TYPE U_Union :
UNION
	INT_	: INT;
	BOOL_	: BOOL;
	UDINT_	: UDINT;
	STRING_	: STRING;
	REAL_	: REAL;
END_UNION
END_TYPE

(* stored: Version 1.1.0.1, ProductVersion 3.1.4024.12
   DUT U_Union: Id {33ff04a7-14e0-4b70-9de6-628158e05b37} *)
